GLOBALCONSTANTS Hutschienenmoped_XL_DO (* Global constants *)
  (* Standard: 61499-1 *)
  (* Version 1.0, 2024-01-25, franz *)
  VAR_GLOBAL CONSTANT
    Output_Q1 : USINT := 1;
    Output_Q2 : USINT := 2;
    Output_Q3 : USINT := 3;
    Output_Q4 : USINT := 4;
    Output_Q5 : USINT := 5;
    Output_Q6 : USINT := 6;
    Output_Q7 : USINT := 7;
    Output_Q8 : USINT := 8;
    Output_Q9 : USINT := 9;
  END_VAR
END_GLOBALCONSTANTS
